Universal Robots PolyScope program: vt1working version.urp

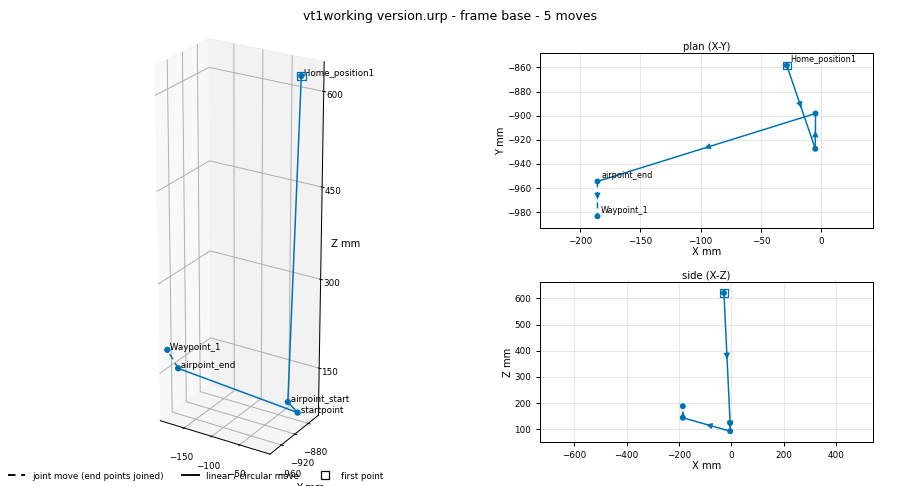
[picture p0: tool path of vt1working version.urp in frame base, 5 of 5 moves have a stored position in this frame; points joined in program order, loops and branches not executed]
Program vt1working version (installation=default directory=/programs/usbdisk/new folder_1 createdIn=5.12.2.1101534 lastSavedIn=5.12.2.1101534 robotSerialNumber=20225202267)
Calibrated DH parameters: a=[0.000057, -0.560337, -0.56987, 0.000044, 0.000023, 0]; d=[0.180974, -304.223407, 295.067386, 9.330269, 0.119831, 0.115671]; alpha=[1.570416, 0.000812, 0.004616, 1.569457, -1.570316, 0]; deltaTheta=[0, -0.415128, 6.624286, 0.074029, 0.000002, -0.000001]
Robot Program (runOnlyOnce=true)
  Folder setup
    Script: open=socket_open("192.168.0.56",50000)
    Loop While (checkContinuously=false) expression=open == False
      Script: open=socket_open("192.168.0.56",50000)
    start_code := [0,0]
    act_current := 0
    act_voltage := 0
    act_wirefeed := 0
    act_gasflow := 0
    current := ""
    voltage := ""
    wirefeed := ""
    gasflow := ""
    continuous := True
    Startcollecting := False
  Loop While (checkContinuously=false) expression=continuous
    Wait Condition expression=start_code[1]==1
    MoveJ speed 60 deg/s, acceleration 80 deg/s^2 (useActiveTCP=false) feature=Base
      Waypoint Home_position1: TCP in base x=-28.623 y=-858.474 z=620.531 mm, rx=0.0156 ry=2.9861 rz=-0.6593 rad; joints [-80.269, -101.512, -89.398, -53.769, 90.666, 10.501] deg
    MoveL speed 250 mm/s, acceleration 1200 mm/s^2 (useActiveTCP=true) feature=Base
      Waypoint airpoint_start: TCP in base x=-5.041 y=-927.434 z=124.466 mm, rx=-1.7687 ry=1.8423 rz=0.7398 rad; joints [-78.015, -108.725, -80.253, -78.667, 88.042, 11.578] deg; TCP offset x=0.754 y=-2.491 z=438.568 mm, rx=-0.6235 ry=-0.6001 rz=-1.4503 rad
    MoveL speed 250 mm/s, acceleration 1200 mm/s^2 (useActiveTCP=true) feature=Base
      Waypoint startpoint: TCP in base x=-4.822 y=-898.2 z=93.049 mm, rx=-1.702 ry=1.8293 rz=0.7677 rad; joints [-78.025, -109.176, -82.12, -79.361, 88.717, 13.424] deg
    Script: socket_send_int(3)
    Wait Condition expression=start_code[1]==2
    Script: Startcollecting= True
    URCap MigaWeld (Migaweld, Smooth Robotics ApS) dataModel(id_key=0, tag_version=Version1_1, enable_start_button=true, node_defined=true)
      SuppressedNode
        MoveJ speed 60 deg/s, acceleration 80 deg/s^2 (useActiveTCP=false) feature=Base
          Waypoint Home_position1: TCP in base x=443.981 y=-399.736 z=631.41 mm, rx=0.1259 ry=2.9193 rz=-0.8661 rad; joints [-19.194, -75.001, -112.928, -65.9, 60.614, 71.458] deg
      SuppressedNode
        Wait DigitalInput pin=digital_in[1]; digitalValue=1
      URCap SpeedSlider (Migaweld, Smooth Robotics ApS) dataModel(set_speed=true)
      URCap WeldItem (Migapath, Smooth Robotics ApS) dataModel(MigaPathtitle_key=WeldItem_1)
        URCap Weld seam (Migapath, Smooth Robotics ApS) dataModel(dataModelVersion=1, programVersion=1, travelSpeed=6.0, amplitude=1.4, titleKey=Weld seam, freq=1.5)
          SuppressedNode
            URCap AirPoint (Migapath, Smooth Robotics ApS) dataModel(title_key=Airpoint, jump_visible=true, pose_has_been_offset=false, Pose(key=move_pose_key, Position(key=posePosition, Length(key=X value=0.487428 unit=M), Length(key=Y value=-0.733495 unit=M), Length(key=Z value=0.144507 unit=M)), Rotation(key=poseRotation, Angle(key=RX value=-1.935447 unit=RAD), Angle(key=RY value=1.929826 unit=RAD), Angle(key=RZ value=0.435421 unit=RAD))), JointPositions(key=move_joint_key, JointPosition(key=[1], Angle(key=pos value=-0.655383 unit=RAD)), JointPosition(key=[2], Angle(key=pos value=-1.629773 unit=RAD)), JointPosition(key=[3], Angle(key=pos value=-1.776107 unit=RAD)), JointPosition(key=[4], Angle(key=pos value=-1.068963 unit=RAD)), JointPosition(key=[5], Angle(key=pos value=1.379737 unit=RAD)), JointPosition(key=[6], Angle(key=pos value=0.880011 unit=RAD))))
          URCap AirPoint (Migapath, Smooth Robotics ApS) dataModel(title_key=Startpoint, pose_has_been_offset=false, Pose(key=move_pose_key, Position(key=posePosition, Length(key=X value=-0.004871 unit=M), Length(key=Y value=-0.898179 unit=M), Length(key=Z value=0.093097 unit=M)), Rotation(key=poseRotation, Angle(key=RX value=-1.701912 unit=RAD), Angle(key=RY value=1.829321 unit=RAD), Angle(key=RZ value=0.767654 unit=RAD))), JointPositions(key=move_joint_key, JointPosition(key=[1], Angle(key=pos value=-1.361809 unit=RAD)), JointPosition(key=[2], Angle(key=pos value=-1.905448 unit=RAD)), JointPosition(key=[3], Angle(key=pos value=-1.433262 unit=RAD)), JointPosition(key=[4], Angle(key=pos value=-1.385119 unit=RAD)), JointPosition(key=[5], Angle(key=pos value=1.548436 unit=RAD)), JointPosition(key=[6], Angle(key=pos value=0.23429 unit=RAD))))
          URCap Arc On (Migaweld, Smooth Robotics ApS) dataModel(arcOnWaitTime=0.0)
          URCap Paths: (Migapath, Smooth Robotics ApS)
            URCap Welding path (Migapath, Smooth Robotics ApS) dataModel(selectedPathType=Linear, useShared=true, titleKey=Linear_1, selectedPattern=None, end_has_been_offset=false, Pose(key=endPose, Position(key=posePosition, Length(key=X value=-0.187598 unit=M), Length(key=Y value=-0.891579 unit=M), Length(key=Z value=0.093344 unit=M)), Rotation(key=poseRotation, Angle(key=RX value=-1.702119 unit=RAD), Angle(key=RY value=1.829246 unit=RAD), Angle(key=RZ value=0.767533 unit=RAD))), JointPositions(key=endJoint, JointPosition(key=[1], Angle(key=pos value=-1.566468 unit=RAD)), JointPosition(key=[2], Angle(key=pos value=-1.921097 unit=RAD)), JointPosition(key=[3], Angle(key=pos value=-1.412694 unit=RAD)), JointPosition(key=[4], Angle(key=pos value=-1.384113 unit=RAD)), JointPosition(key=[5], Angle(key=pos value=1.546795 unit=RAD)), JointPosition(key=[6], Angle(key=pos value=0.029516 unit=RAD))))
          URCap Arc Off (Migaweld, Smooth Robotics ApS) dataModel(arcOffWaitTime=0.5)
          SuppressedNode
            URCap AirPoint (Migapath, Smooth Robotics ApS) dataModel(title_key=Airpoint, pose_has_been_offset=false, Pose(key=move_pose_key, Position(key=posePosition, Length(key=X value=0.449835 unit=M), Length(key=Y value=-0.711698 unit=M), Length(key=Z value=0.167888 unit=M)), Rotation(key=poseRotation, Angle(key=RX value=-1.961448 unit=RAD), Angle(key=RY value=1.934564 unit=RAD), Angle(key=RZ value=0.351219 unit=RAD))), JointPositions(key=move_joint_key, JointPosition(key=[1], Angle(key=pos value=-0.650033 unit=RAD)), JointPosition(key=[2], Angle(key=pos value=-1.506743 unit=RAD)), JointPosition(key=[3], Angle(key=pos value=-1.888574 unit=RAD)), JointPosition(key=[4], Angle(key=pos value=-1.019091 unit=RAD)), JointPosition(key=[5], Angle(key=pos value=1.361404 unit=RAD)), JointPosition(key=[6], Angle(key=pos value=0.880223 unit=RAD))))
      SuppressedNode
        MoveJ speed 60 deg/s, acceleration 80 deg/s^2 (useActiveTCP=false) feature=Base
          Waypoint Home_position1: TCP in base x=443.981 y=-399.736 z=631.41 mm, rx=0.1259 ry=2.9193 rz=-0.8661 rad; joints [-19.194, -75.001, -112.928, -65.9, 60.614, 71.458] deg
    Script: Startcollecting= False
    Script: socket_send_int(4)
    MoveL speed 250 mm/s, acceleration 1200 mm/s^2 (useActiveTCP=true) feature=Base
      Waypoint airpoint_end: TCP in base x=-185.501 y=-954.485 z=144.333 mm, rx=-1.8199 ry=1.9048 rz=0.6823 rad; joints [-89.237, -108.365, -80.276, -73.847, 87.912, 0.313] deg; TCP offset x=0.754 y=-2.491 z=438.568 mm, rx=-0.6235 ry=-0.6001 rz=-1.4503 rad
    MoveJ speed 60 deg/s, acceleration 80 deg/s^2 (useActiveTCP=true) feature=Base
      Waypoint Waypoint_1: TCP in base x=-185.501 y=-983.434 z=188.425 mm, rx=-1.82 ry=1.9048 rz=0.6822 rad; joints [-89.263, -110.704, -72.649, -79.129, 87.927, 0.264] deg
Thread Thread_1 (runOnlyOnce=false)
  Script: act_current=read_input_integer_register(5)
  Script: act_voltage=read_input_integer_register(6)
  Script: act_wirefeed=read_input_integer_register(5)
  Script: act_gasflow=read_input_integer_register(5)
  Script: start_code=socket_read_ascii_float(1)
  If Startcollecting== True (checkContinuously=true)
    Script: current=str_cat(to_str(act_current),",")
    Script: voltage=str_cat(to_str(act_voltage),",")
    Script: wirefeed=str_cat(to_str(act_wirefeed),",")
    Script: gasflow=str_cat(to_str(act_gasflow),",")
    Script: socket_send_string(str_cat(str_cat(current,voltage),str_cat(wirefeed,gasflow)))
  If start_code[1]==5
    Script: continuous= False
    Halt
  Wait Sleep waitTime=0.01
